SUBAPPLICATION Ventilsteuerung_Uebung_014 (* Container (visible/invisible) *)
  (* Standard: 61499-2 *)
  (* Version 1.0, 2023-10-23, franz *)
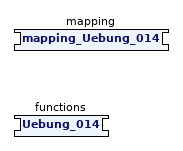
  SUBAPPS
    mapping : mapping_Uebung_014;
    functions : Uebung_014;
  END_SUBAPPS
END_SUBAPPLICATION
